FUNCTION Convert_UINT_TO_SINT : Hresult
VAR_INPUT
	in : UINT;
	out : REFERENCE TO SINT;
END_VAR
VAR
	converted : SINT;
END_VAR
VAR CONSTANT
	INCOMPATIBLE : HRESULT := 16#9811070E;
END_VAR

converted := UINT_TO_SINT(in);

IF (SINT_TO_UINT(converted) <> in) THEN
	Convert_UINT_TO_SINT := INCOMPATIBLE;
	RETURN;
END_IF

out := converted;

END_FUNCTION

(* stored: Version 1.1.0.1, ProductVersion 3.1.4024.12
   POU Convert_UINT_TO_SINT: Id {e482e318-d545-440d-84e6-d04a4047a964}, SpecialFunc None *)
